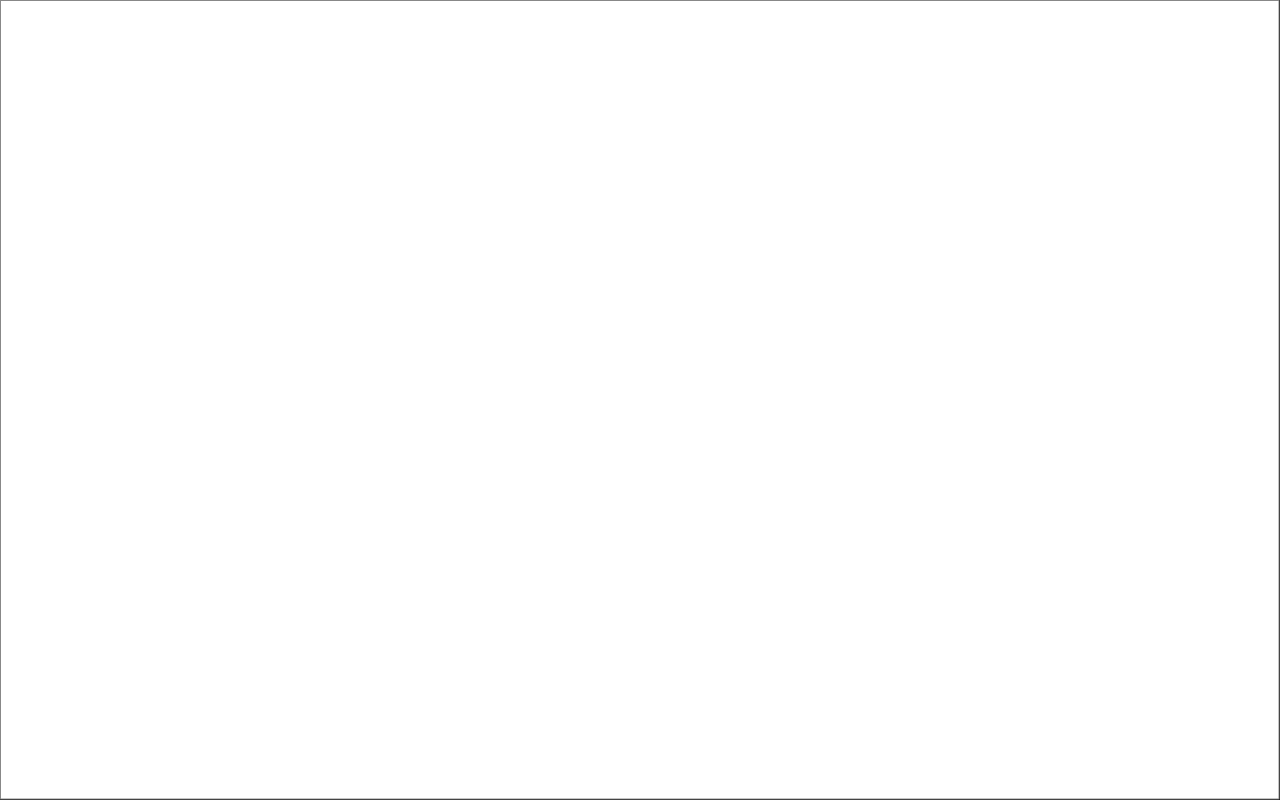
VISUALIZATION Automatic  // 1280x800
    Rectangle (0,0 1280x800)
END_VISUALIZATION

(* stored: Version 1.1.0.1, ProductVersion 3.1.4024.5
   Visu Automatic: Id {17973cfd-bff5-454c-9e28-145b8ffd4d4a} *)
